// vecB=VecA*num
FUNCTION vecMultiNum : BOOL
VAR_IN_OUT CONSTANT
	vecA :ARRAY[*] OF LREAL;
END_VAR

VAR_INPUT
	num :LREAL;
END_VAR

VAR_IN_OUT
	vecB : ARRAY[*] OF LREAL;
END_VAR
VAR
	m :DINT;
	i :DINT;
END_VAR

m:=UPPER_BOUND(vecA,1);

FOR i:=1 TO m DO
		vecB[i]:=num*vecA[i];
END_FOR

END_FUNCTION

(* stored: Version 1.1.0.1, ProductVersion 3.1.4024.12
   POU vecMultiNum: Id {3666d1a2-525d-470a-9200-d5986843e7ee}, SpecialFunc None *)
